// TIA Portal V16 export
// export: Created 2024-12-03T15:41:43.3665087Z, ExportSetting WithDefaults, DisplayName Totally Integrated Automation Portal, DisplayVersion V16 Update 6, DisplayName TIA Portal Version Control Interface, DisplayVersion V16 Update 2, DisplayName TIA Portal Openness, DisplayVersion V16 Update 6, DisplayName TIA Portal Teamcenter Gateway, DisplayVersion V16, DisplayName SINAMICS Startdrive Advanced, DisplayVersion V16 Update 5, DisplayName SINAMICS Startdrive G130, G150, S120, S150, SINAMICS MV, S210, DisplayVersion V16 Update 5, DisplayName SINAMICS Startdrive G110M, G120, G120C, G120D, G120P, G115D, DisplayVersion V16 Update 5, DisplayName STEP 7 Professional, DisplayVersion V16 Update 6, DisplayName STEP 7 Safety, DisplayVersion V16, DisplayName WinCC Advanced / Unified PC, DisplayVersion V16 Update 6
FUNCTION_BLOCK "TrafficController_INTERSECT_SENDING_FB"   // FB36, SCL
{ S7_Optimized_Access := 'TRUE' }
VERSION : 0.1
// intersection receives from one section and can sent to other 3 sections
// stored: AutoNumber true, IsIECCheckEnabled false, IsRetainMemResEnabled false, MemoryReserve 100, SetENOAutomatically false, UDAEnableTagReadback false
   VAR_INPUT
      I_Option : Int;
      I_IntersectionConveyor : "Conveyor_UDT";
      I_Option_1_Settings { ExternalAccessible := 'False'; ExternalVisible := 'False'; ExternalWritable := 'False'} : "Intersection";   // Intersection settings for option 1 (no split executed)
      I_Option_2_Settings { ExternalAccessible := 'False'; ExternalVisible := 'False'; ExternalWritable := 'False'} : "Intersection";   // Intersection settings for option 2 (split executed)
      I_Option_3_Settings { ExternalAccessible := 'False'; ExternalVisible := 'False'; ExternalWritable := 'False'} : "Intersection";   // Intersection settings for option 2 (split executed)
      I_Option_4_Settings { ExternalAccessible := 'False'; ExternalVisible := 'False'; ExternalWritable := 'False'} : "Intersection";   // Intersection settings for option 2 (split executed)
      I_Option_5_Settings { ExternalAccessible := 'False'; ExternalVisible := 'False'; ExternalWritable := 'False'} : "Intersection";   // Intersection settings for option 2 (split executed)
      I_Option_6_Settings { ExternalAccessible := 'False'; ExternalVisible := 'False'; ExternalWritable := 'False'} : "Intersection";   // Intersection settings for option 2 (split executed)
   END_VAR
   VAR_IN_OUT
      IO_SendingConveyor : "Conveyor_UDT";
      IO_IntersectionSettings : "Intersection";
   END_VAR
   VAR
      option : Int;
      OptionsSaved : Bool;
   END_VAR
BEGIN
   #IO_SendingConveyor.Cmd.Accumulate.Acc_TC_1 := TRUE;

   REGION CHECK TO TRANSFER SETTINGS

       IF #IO_SendingConveyor.Status.RequestForSending
           AND #I_IntersectionConveyor.Status.Empty THEN

           CASE #I_Option OF
               1:
                   #IO_IntersectionSettings := #I_Option_1_Settings;
               2:
                   #IO_IntersectionSettings := #I_Option_2_Settings;
               3:
                   #IO_IntersectionSettings := #I_Option_3_Settings;
               4:
                   #IO_IntersectionSettings := #I_Option_4_Settings;
               5:
                   #IO_IntersectionSettings := #I_Option_5_Settings;
               6:
                   #IO_IntersectionSettings := #I_Option_6_Settings;
           END_CASE;


       END_IF;

   END_REGION

   REGION TURN OFF ACCUMULATION OF SENDING CONV

       IF #I_IntersectionConveyor.Status.Empty
           AND #IO_SendingConveyor.Status.RequestForSending THEN
           //AND #I_SendingConveyor.TrackingStat.Current.PLC_Dest >= 0 THEN
           #IO_SendingConveyor.Cmd.Accumulate.Acc_TC_1 := FALSE;
       END_IF;

   END_REGION
END_FUNCTION_BLOCK
